FUNCTION_BLOCK F_BYTE_BCD_TO_USINT (* convert BYTE  Binary Coded Decimal to USINT *)
  (* Standard: 61131-3; Classification: standard type conversion function; Description: Copyright (c) 2013 TU Wien ACIN This program and the accompanying materials are made available under the terms of the Eclipse Public License 2.0 which is available at https://www.eclipse.org/legal/epl-2.0/ SPDX-License-Identifier: EPL-2.0 *)
  (* Version 1.0, 2013-09-07, Monika Wenger, TU Wien ACIN *)
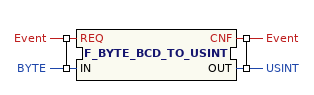
  EVENT_INPUT
    REQ WITH IN; (* Service Request *)
  END_EVENT
  EVENT_OUTPUT
    CNF WITH OUT; (* Confirmation of Requested Service *)
  END_EVENT
  VAR_INPUT
    IN : BYTE; (* input value *)
  END_VAR
  VAR_OUTPUT
    OUT : USINT; (* output value *)
  END_VAR
  (* Service APPLICATION/RESOURCE: convert BYTE  Binary Coded Decimal to USINT *)
END_FUNCTION_BLOCK
